FUNCTION F_HomeOffsetCalc : LREAL
VAR_INPUT
	CurrentOffset: LREAL;
	CurrentPosition: LREAL;
	HomeSearchDirection: MC_Direction;
END_VAR

IF HomeSearchDirection = MC_Direction.positive THEN
	F_HomeOffsetCalc := -F_RoundLreal(ABS(CurrentPosition - CurrentOffset),2);
	
ELSIF HomeSearchDirection = MC_Direction.negative THEN
	F_HomeOffsetCalc := F_RoundLreal(ABS(CurrentPosition - CurrentOffset),2);
	
ELSE
	F_HomeOffsetCalc := CurrentOffset;
	
END_IF

END_FUNCTION

(* stored: Version 1.1.0.1
   POU F_HomeOffsetCalc: Id {ad8953b8-d17f-41b2-83c9-9901a22a0b46}, SpecialFunc None *)
